// TIA Portal V20 export
VAR_GLOBAL   // PLC tag table "LGR_Const_Interface_Validation"
END_VAR
VAR_GLOBAL CONSTANT   // user constants
   INVALID_PROTOCOL : UInt := 100;
   INVALID_CMD : UInt := 101;
   INVALID_SRC : UInt := 102;
   INVALID_DST : UInt := 103;
   INVALID_DUPLICATED : UInt := 104;
   INVALID_TASK_WORKID : UInt := 200;
   INVALID_TASK_TASKID : UInt := 201;
   INVALID_TASK_WORKCELL : UInt := 202;
   INVALID_TASK_TYPE : UInt := 203;
   INVALID_TASK_POSX : UInt := 301;
   INVALID_TASK_POSY : UInt := 302;
   INVALID_TASK_POSZ : UInt := 303;
   INVALID_TASK_POSG : UInt := 304;
   INVALID_TASK_BLENDUP : UInt := 310;
   INVALID_TASK_BLENDDOWN : UInt := 311;
   INVALID_TASK_ITEM_CODE : UInt := 501;
   INVALID_TASK_ITEM_COUNT : UInt := 502;
   INVALID_UNDEFINED : UInt := 900;
   VALID_TASK_DATA : UInt := 1;
   INVALID_TASK_DRAGOUT_HEIGHT : UInt := 321;
   INVALID_TASK_DRAGOUT_DIST : UInt := 322;
   INVALID_TASK_DRAGOUT_DIR : UInt := 323;
   INVALID_TASK_DRAGIN_HEIGHT : UInt := 331;
   INVALID_TASK_DRAGIN_DIST : UInt := 332;
   INVALID_TASK_DRAGIN_DIR : UInt := 333;
   INVALID_TASK_DRAGOUT_USE : UInt := 320;
   INVALID_TASK_DRAGIN_USE : UInt := 330;
   INVALID_TASK_GRIP_DELTA : UInt := 340;
   INVALID_CELL_ID_EMPTY : UInt := 401;
   INVALID_STATION_RANGE_X : UInt := 411;
   INVALID_CELL_SECTION : UInt := 420;
   INVALID_CELL_RANGE_X : UInt := 421;
   INVALID_CELL_RANGE_Y : UInt := 422;
   INVALID_STATION_RANGE_Y : UInt := 412;
   INVALID_STATION_NO_RESISTRY : UInt := 419;
   INVALID_CELL_NO_RESISTRY : UInt := 429;
   INVALID_AREA_UNDEFINE : UInt := 409;
   INVALID_STATION_RANGE_Z : UInt := 413;
   INVALID_STATION_SECTION : UInt := 410;
   INVALID_CELL_RANGE_Z : UInt := 423;
   INVALID_CELL_USE : UInt := 428;
   INVALID_STATION_USE : UInt := 418;
   INVALID_BUFFERFULL : UInt := 110;
   INVALID_CELL_POSZ : UInt := 305;
END_VAR
